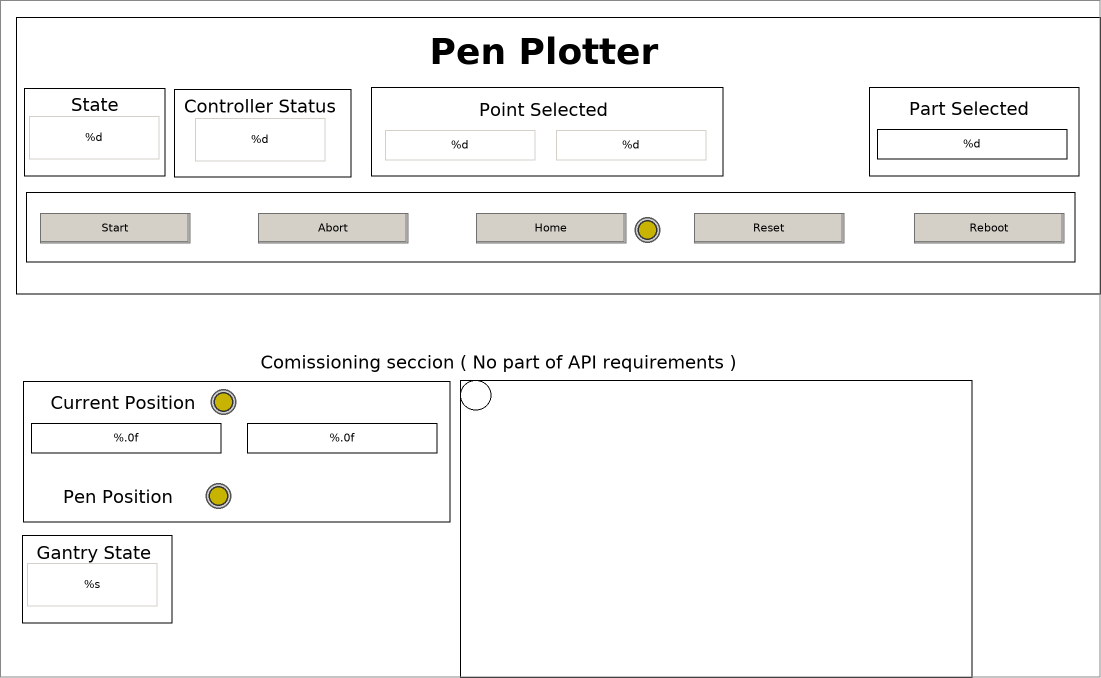
VISUALIZATION HMI  // 1101x678
    RoundedRectangle (16,17 1085x277)
    RoundedRectangle (23,381 427x141)
    Rectangle (247,423 190x30), "%.0f", text variable: MAIN.my_gantry.sts.position.y
    Rectangle (31,423 190x30), "%.0f", text variable: MAIN.my_gantry.sts.position.x
    Lamp1 (205,387 37x30), variable: MAIN.my_gantry.sts.at_position, style: Lamp-Lamp1-Yellow
    Label (28,388 190x30), "Current Position"
    RoundedRectangle (371,87 352x89)
    Textfield (385,130 150x30), "%d", text variable: MAIN.api_fromHMI.stsPointSelected[0]
        OnMouseDown: write the text variable via InputWithLimits, min 0, max 1000, title 'Target Position X'
    Textfield (556,130 150x30), "%d", text variable: MAIN.api_fromHMI.stsPointSelected[1]
        OnMouseDown: write the text variable via InputWithLimits, min 0, max 1000, title 'Target Position X'
    Label (384,95 319x30), "Point Selected"
    RoundedRectangle (24,88 141x88)
    Textfield (29,116 130x43), "%d", text variable: MAIN.api_toHMI.stsState
    Label (28,90 134x30), "State"
    RoundedRectangle (26,192 1049x70)
    Button (914,213 150x30), "Reboot"
        tap MAIN.api_fromHMI.stsReboot
    Button (40,213 150x30), "Start"
        tap MAIN.api_fromHMI.cmdStart p1329445385=TRUE
    Button (258,213 150x30), "Abort"
        tap MAIN.api_fromHMI.cmdAbort p1329445385=TRUE
    Button (476,213 150x30), "Home"
        tap MAIN.api_fromHMI.cmdHome
    Button (694,213 150x30), "Reset"
        tap MAIN.api_fromHMI.cmdReset p1329445385=TRUE
    Label (25,22 1038x59), "Pen Plotter"
    RoundedRectangle (174,89 177x88)
    Textfield (195,118 130x43), "%d", text variable: MAIN.api_toHMI.stsState
    Label (178,93 164x27), "Controller Status"
    Label (26,349 945x27), "Comissioning seccion ( No part of API requirements )"
    RoundedRectangle (869,87 210x89)
    Rectangle (877,129 190x30), "%d", text variable: MAIN.api_toHMI.stsPartSelected
    Label (874,94 190x30), "Part Selected"
    Lamp1 (200,481 37x30), variable: MAIN.cmd_penAdvance, style: Lamp-Lamp1-Yellow
    Label (23,482 190x30), "Pen Position"
    Label (26,537 134x30), "State"
    RoundedRectangle (22,535 150x88)
    Textfield (27,563 130x43), "%s", text variable: MAIN.my_gantry.sts.state_text
    Label (27,538 134x30), "Gantry State"
    Lamp1 (629,215 37x30), variable: MAIN.my_gantry.sts.all_homed, style: Lamp-Lamp1-Yellow
    Rectangle (460,380 512x298)
    Ellipse (460,380 31x30)
        p3560616238: MAIN.my_gantry.sts.position.x
        p2738717112: MAIN.my_gantry.sts.position.y
END_VISUALIZATION

(* stored: Version 1.1.0.1, ProductVersion 3.1.4024.13
   Visu HMI: Id {b9198251-3c00-4234-8868-5c45d5f7d13c} *)
